// TIA Portal V17 export
// export: Created 2024-09-02T12:50:40.6586702Z, ExportSetting WithDefaults, DisplayName Totally Integrated Automation Portal, DisplayVersion V17, DisplayName TIA Portal Openness, DisplayVersion V17, DisplayName TIA Portal Version Control Interface, DisplayVersion V17, DisplayName STEP 7 Professional, DisplayVersion V17, DisplayName STEP 7 Safety, DisplayVersion V17, DisplayName WinCC Professional, DisplayVersion V17
TYPE "Aveva_Scanner_Result"
// stored: IsFailsafeCompliant false
   STRUCT
      Status { ExternalWritable := 'False'} : Array[0..7] of Bool;   // %X0-Work Finished NOK/%X1 Work Finished OK /%X2 Work Bypassed /%X3 Work Interrupted
      RetryPerformed { ExternalWritable := 'False'} : Int;   // Number of retry
      Scanner_Result { ExternalWritable := 'False'} : String[25];   // traceability data
   END_STRUCT;
END_TYPE
